PROGRAM P_Time
VAR
    fbSystemTime : GETSYSTEMTIME;
	fbSystemTime2 : FB_GetSystemTime;
    timeAsFileTime : T_FILETIME;
    timeAsDT : DT;
	actual_date_meawhile :DT;
	s_time_mainscreen	:WSTRING(80);
	tonBreakTurnOff 	:TON;
END_VAR

tonBreakTurnOff(IN:=gvl_cfg.bBreakReset,PT:=T#5S);
fbSystemTime2(bEnable:=TRUE);
fbSystemTime(
    timeLoDW => timeAsFileTime.dwLowDateTime,
    timeHiDW => timeAsFileTime.dwHighDateTime 
);
(*timeAsDT := FILETIME_TO_DT(timeAsFileTime);
actual_date_meawhile:=timeAsDT;
actual_date_meawhile := actual_date_meawhile + T#2H;
s_time_mainscreen := DT_TO_WSTRING(actual_date_meawhile);
s_time_mainscreen := WRIGHT(s_time_mainscreen, WLEN(s_time_mainscreen) - 3);
gvl_his.s_time_mainscreen:=s_time_mainscreen;
gvl_cfg.wsRightTime:=WRIGHT(s_time_mainscreen,8);*)
timeAsDT :=fbSystemTime2.dtActTime;
actual_date_meawhile:=timeAsDT;
s_time_mainscreen := DT_TO_WSTRING(actual_date_meawhile);
s_time_mainscreen := WRIGHT(s_time_mainscreen, WLEN(s_time_mainscreen) - 3 );
gvl_gauge.s_time_mainscreen:=s_time_mainscreen;


IF gvl_cfg.sRightTime = gvl_cfg.tbreakTime_1 OR gvl_cfg.sRightTime = gvl_cfg.tbreakTime_2 THEN
	gvl_cfg.bBreakReset:=TRUE;
END_IF

IF tonBreakTurnOff.Q THEN
	gvl_cfg.bBreakReset:=FALSE;
END_IF

END_PROGRAM

(* stored: Version 1.1.0.1, ProductVersion 3.1.4026.13, FileIdentifier 3179d592f69638fc7349b98f8b7d6c29349084ee, FileSignature 7c21e43cae7ac6f7d6e0a53707454243a3663b8a213ec0b8c39cc49dfe000ffd42002ff45ad423629a7dda39f3d5225a13d704215154275f1e7dcf401f5a054151521488afd2df554930e8507dc82739329f1b1426501252674dd1647d0691ceec051483b3e73861d292cbf26c64f44ceef1af47b4483afcd48ecdb4d8e060d53113e6d3026c7bb8a20082d64fe59efb46e69b7deda16af60275e4b8a858b1472b16d392714e9cfd72b62e91aa54e6c8bace39f08598a5062c780e2337a909e02a02df9188bc3669de5990719f01baa419bb5333906e195c4817914adf543a2b6ba89e27d4adb80b8c5626a822b20daa643c665305ae76d7f397f25d34f10dce
   POU P_Time: Id {aa9264fc-39ea-42a6-97ad-99c5a5cff593}, SpecialFunc None *)
